// TwinCAT 3 PLC project TEST_ADS_PC
// ProgramVersion: 3.1.4023.0
// libraries:
//   Tc2_Standard, * (Beckhoff Automation GmbH)
//   Tc2_System, * (Beckhoff Automation GmbH)
//   Tc3_Module, * (Beckhoff Automation GmbH)
// project tree:
//   / PlcTask.TcTTO
//   POUs/ MAIN.TcPOU
// real-time tasks:
//   TASK PlcTask1: cycle T#10ms, priority 21, ADS port 351
//   TASK Task 3: cycle T#10ms, priority 1, ADS port 351
// I/O:
//   DEVICE Device 2 (EtherCAT), AmsNetId 192.168.102.2.3.1
//     Box 1 (EL6695-0002) [EL6695 EtherCAT Bridge terminal (Secondary)]
// variable links:
//   Task 3 <-> Device 2 (EtherCAT)/Box 1 (EL6695-0002)
//     Inputs/VarInPlc <-> IO Inputs/VarInRobot
//     Outputs/VarOutPlc <-> IO Outputs/VarOutRobot

CONFIGURATION TEST_ADS_PC
    RESOURCE PLC ON TwinCAT3
        TASK PlcTask(INTERVAL := T#10ms, PRIORITY := 21);
        PROGRAM MAIN WITH PlcTask : MAIN;
    END_RESOURCE
END_CONFIGURATION

// ---- POUs/MAIN.TcPOU
PROGRAM MAIN
VAR
	ROBOTVar AT %MD0 : DWORD;
	PCVar AT %MD1 : DWORD;
	TP_1		: TP;
	TOGGEL: BOOL;
END_VAR

TOGGEL := NOT TOGGEL;
TP_1( IN := TOGGEL, PT := T#100ms);
IF (TP_1.Q = 0) THEN
	ROBOTVar := ROBOTVar + 1;
END_IF

END_PROGRAM
